TYPE "PosList"
VERSION : 0.1
   STRUCT
      List : Array[0..39] of Struct
         Pos : DInt;
         Vel : Int;
      END_STRUCT;
   END_STRUCT;

END_TYPE

